// TIA Portal project "PROJECT DRIVES" (V17)

(* hardware
DEVICE "S7-1200 station_1"  S7-1200 Station
   slot 0: "Rack_0"  S7-1200 Rack  Rack  V1.0
   slot 1: "PLC_1"  CPU 1214C DC/DC/DC  6ES7 214-1AG40-0XB0  V4.2
DEVICE "HMI_1"  KTP700 Basic PN
   slot 0: "HMI_1"  KTP700 Basic PN  6AV2 123-2GB03-0AX0  15.0.0.0
   slot 1: "HMI_RT_1"  KTP700 Basic PN  6AV2 123-2GB03-0AX0  15.0.0.0
   slot 5: "HMI_1.IE_CP_1"  PROFINET Interface  15.0.0.0
      slot 1: "PROFINET Interface_1"  PROFINET Interface
         slot 1: "Port_1"  Port
DEVICE "ET 200SP station_1"  ET 200SP-Station
   slot 0: "Rack_0"  Rack  6ES5 710-8MAx1
   slot 0: "IO device_1"  IM 155-6 PN/2 HF  6ES7 155-6AU01-0CN0  V4.2
   slot 1: "DQ 8x24VDC/0.5A HF_1"  DQ 8x24VDC/0.5A HF  6ES7 132-6BF00-0CA0  V2.0
      slot 1: "DQ 8x24VDC/0.5A HF_1"  DQ 8x24VDC/0.5A HF
   slot 2: "DQ 8x24VDC/0.5A HF_2"  DQ 8x24VDC/0.5A HF  6ES7 132-6BF00-0CA0  V2.0
      slot 1: "DQ 8x24VDC/0.5A HF_2"  DQ 8x24VDC/0.5A HF
   slot 3: "DI 8x24VDC HF_1"  DI 8x24VDC HF  6ES7 131-6BF00-0CA0  V2.0
      slot 1: "DI 8x24VDC HF_1"  DI 8x24VDC HF
   slot 4: "DI 8x24VDC HF_2"  DI 8x24VDC HF  6ES7 131-6BF00-0CA0  V2.0
      slot 1: "DI 8x24VDC HF_2"  DI 8x24VDC HF
   slot 5: "DI 8x24VDC HF_3"  DI 8x24VDC HF  6ES7 131-6BF00-0CA0  V2.0
      slot 1: "DI 8x24VDC HF_3"  DI 8x24VDC HF
   slot 6: "Server module_1"  Server module  6ES7 193-6PA00-0AA0  V1.1
      slot 1: "Server module_1"  Server module
   slot 127: "BA 2xRJ45"  BA 2xRJ45  6ES7 193-6AR00-0AA0  V0.0
      slot 1: "Port_1"  X1 P1 R  6ES7 193-6AR00-0AA0  V0.0
      slot 2: "Port_2"  X1 P2 R  6ES7 193-6AR00-0AA0  V0.0
DEVICE "SCALANCE X005"  SCALANCE X-Station
   slot 0: "SCALANCE X rack"  Rail
   slot 0: "Switch_1"  6GK5 005-0BA00-1AB2  V1.0
DEVICE "GSD device_1"  GSD.Device.PN
   slot 0: "Rack"  Rack  V1.0
   slot 0: "drivexb14fe3"  SINAMICS G120 CU250S-2 PN Vector V4.7  6SL3 246-0BA22-1FAx  V4.70
      slot 0: "SINAMICS G120 CU250S-2 PN Vector V4.7"  SINAMICS G120 CU250S-2 PN Vector V4.7
      slot 1: "DO VECTOR_1"  DO VECTOR
         slot 0: "Module Access Point"  Module Access Point
      slot 1: "PN-IO"  PN-IO
         slot 1: "Port 1"  Port 1
         slot 2: "Port 2"  Port 2
   slot 2: "Standard telegram 2, PZD-4/4"  Standard telegram 2, PZD-4/4
*)

// ===== PLC "PLC_1"  CPU 1214C DC/DC/DC =====

VAR_GLOBAL   // PLC tag table "Default tag table"
   "SYSTEM ON" AT %M10.0 : Bool;
   "CWT" AT %QW64 : Word;
   "STW" AT %QW66 : Word;
END_VAR

TYPE "HMI"
   STRUCT
      START : Bool;
      STOP : Bool;
      "MOTOR ON" : Bool;
      "MOTOR OFF" : Bool;
   END_STRUCT;
END_TYPE

DATA_BLOCK "HMI_DATA"   // DB1
{ S7_Optimized_Access := 'FALSE' }
VERSION : 0.1
   VAR
      Static_1 : Array[0..4] of Bool;
   END_VAR
BEGIN
END_DATA_BLOCK

// folder: System blocks/Program resources

DATA_BLOCK "IEC_Timer_0_DB"   // DB2
{ S7_Optimized_Access := 'TRUE' }
AUTHOR : Simatic
FAMILY : IEC
NAME : IEC_TMR
VERSION : 1.0
// stored: InstanceOfName IEC_TIMER
"IEC_TIMER"
BEGIN
END_DATA_BLOCK

// folder: (top level)

ORGANIZATION_BLOCK "Main"   // OB1, LAD, ProgramCycle
TITLE = "Main Program Sweep (Cycle)"
{ S7_Optimized_Access := 'TRUE' }
VERSION : 0.1
   VAR_INPUT
      Initial_Call : Bool;   // Initial call of this OB
      Remanence : Bool;   // =True, if remanent data are available
   END_VAR
BEGIN

REGION Network 1
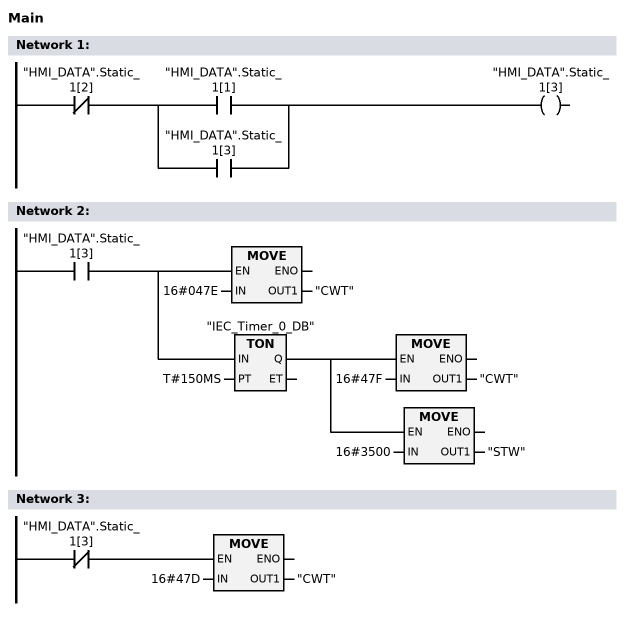
   RUNG wire#powerrail
      I_Contact( "HMI_DATA".Static_1[2] )
      wire#w1
      Contact( "HMI_DATA".Static_1[1] )
      wire#w2
      Coil( "HMI_DATA".Static_1[3] )
   END_RUNG
   RUNG wire#w1
      Contact( "HMI_DATA".Static_1[3] )
   END_RUNG wire#w2
   // the same network as SCL:
   "HMI_DATA".Static_1[3] := NOT "HMI_DATA".Static_1[2] AND ("HMI_DATA".Static_1[1] OR "HMI_DATA".Static_1[3]);
END_REGION

REGION Network 2
   IF "HMI_DATA".Static_1[3] THEN "CWT" := 16#047E; END_IF;
   "IEC_Timer_0_DB".TON(IN := "HMI_DATA".Static_1[3], PT := T#150MS);
   IF "IEC_Timer_0_DB".Q THEN
       "CWT" := 16#47F;
       "STW" := 16#3500;
   END_IF;
END_REGION

REGION Network 3
   RUNG wire#powerrail
      I_Contact( "HMI_DATA".Static_1[3] )
      Move(in := 16#47D, out1 => "CWT")
   END_RUNG
   // the same network as SCL:
   IF NOT "HMI_DATA".Static_1[3] THEN "CWT" := 16#47D; END_IF;
END_REGION
END_ORGANIZATION_BLOCK

(* ===== HMI "HMI_RT_1" =====
system functions are stored by id; their names below are inferred from use
connection "HMI_Connection_1": ETHERNET, SMART_S7_1200_OMS

HMI tags "Default tag table"
   "HMI_DATA_Static_1{1}" : Bool = PLC HMI_DATA.Static_1[1] AT %DB1.DBX0.1, 1 s
   "HMI_DATA_Static_1{2}" : Bool = PLC HMI_DATA.Static_1[2] AT %DB1.DBX0.2, 1 s
   "HMI_DATA_Static_1{4}" : Bool = PLC HMI_DATA.Static_1[4] AT %DB1.DBX0.4, 1 s
   "HMI_DATA_Static_1{0}" : Bool = PLC HMI_DATA.Static_1[0] AT %DB1.DBX0.0, 1 s

screen "Screen_1" 800x480
   Button "Button_1" at 122,107 size 120x55; TextOff 'START'
      on Press: SetBit("HMI_DATA_Static_1{1}")
      on Release: ResetBit("HMI_DATA_Static_1{1}")
   Button "Button_2" at 123,208 size 120x55; TextOff 'STOP'
      on Press: SetBit("HMI_DATA_Static_1{2}")
      on Release: ResetBit("HMI_DATA_Static_1{2}")
*)